Fanuc KAREL source: remote_position.kl

PROGRAM remoteposition
%COMMENT = ' Remote Position'
%NOLOCKGROUP
%NOBUSYLAMP

VAR
	response_file :FILE
	STATUS: INTEGER

	%INCLUDE ../core/core_position

BEGIN
	OPEN FILE response_file ('RW', 'RD:RESPONSE.HTM')
	STATUS = IO_STATUS(response_file)
	IF (STATUS <> 0) THEN
		RETURN
	ENDIF

	CORE_POSITION(response_file)

	CLOSE FILE response_file
END remoteposition
